DATA_BLOCK "Zne02_DB"
{ S7_Optimized_Access := 'TRUE' }
VERSION : 0.1
NON_RETAIN
"Zne02"

BEGIN

END_DATA_BLOCK

